(* LS Electric XG5000 project: PRACTICE3 *)
(* PLC LSPLC *)

PROGRAM NewProgram (* task: 스캔 프로그램 *)
VAR
    ARRAY_TIME : ARRAY[0..2] OF STRING;
    ARRAY_TIME0 : STRING := 'T#';
    ARRAY_TIME2 : STRING := 's';
    FUN : TP;
    PT : TIME;
    TIME_STRING : STRING;
END_VAR
VAR
    _e1 : R_TRIG;
END_VAR

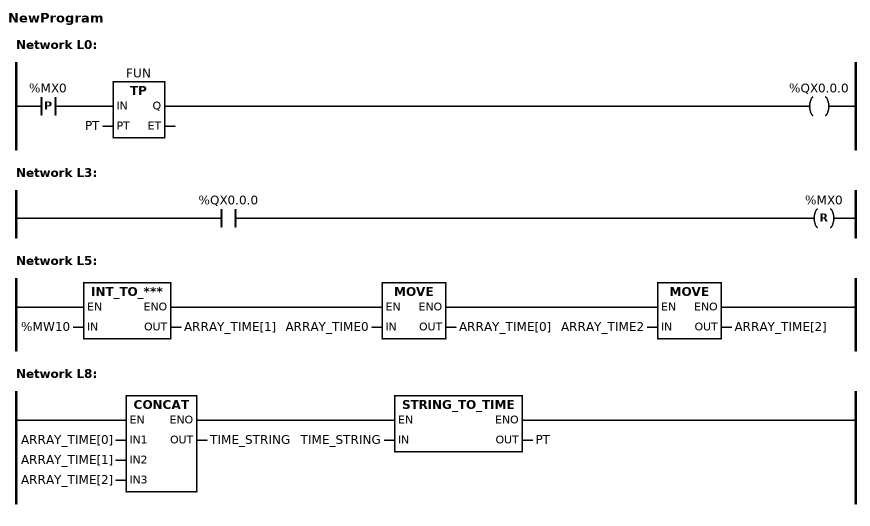
(* Rung L0 *)
_e1(CLK := %MX0);
FUN(IN := _e1.Q, PT := PT);
%QX0.0.0 := FUN.Q;
(* Rung L3 *)
IF %QX0.0.0 THEN %MX0 := FALSE; END_IF;
(* Rung L5 *)
ARRAY_TIME[1] := INT_TO_***(%MW10);
ARRAY_TIME[0] := ARRAY_TIME0;
ARRAY_TIME[2] := ARRAY_TIME2;
(* Rung L8 *)
TIME_STRING := CONCAT(ARRAY_TIME[0], ARRAY_TIME[1], ARRAY_TIME[2]);
PT := STRING_TO_TIME(TIME_STRING);
END_PROGRAM

PROGRAM PRECTICE3 (* task: 스캔 프로그램 *)
VAR
    FUN : TP_UINT;
    RESET : BOOL;
END_VAR
VAR
    _e1 : R_TRIG;
END_VAR

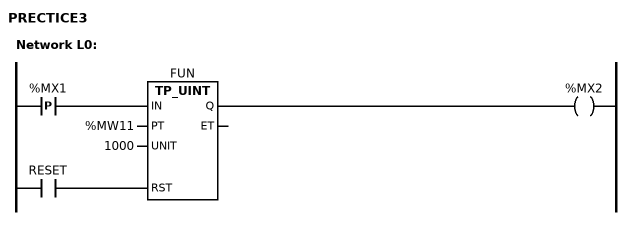
(* Rung L0 *)
_e1(CLK := %MX1);
FUN(IN := _e1.Q, PT := %MW11, UNIT := 1000, RST := RESET);
%MX2 := FUN.Q;
END_PROGRAM